{attribute addProperty BoxType "EK1100-0000-0018"}
{attribute addProperty Id "Beckhoff_EPP2xxxEK1122Beckhoff_EPP2xxxEK1122_0CAC7812157361967"}
{attribute addProperty CRC "2145404589"}
{attribute addProperty SizeInBites "15736"}
{attribute addProperty SizeInBytes "1967"}
TYPE Beckhoff_EPP2xxx_7FE046AD EXTENDS EK1100_179A0949 :
STRUCT
	{attribute addProperty Name "Beckhoff_EPP2xxxEK1122"}
	Beckhoff_EPP2xxxEK1122 : Beckhoff_EPP2xxxEK1122_0CAC7812;
END_STRUCT
END_TYPE

(* stored: Version 1.2.0.0, ProductVersion 3.1.4024.9
   DUT Beckhoff_EPP2xxx_7FE046AD: Id {4e5d2f80-027c-414b-b59a-2bf4eda2cbf7} *)
